// TIA Portal V18 export
TYPE "UDT_HCsDI"
// stored: IsFailsafeCompliant false
   STRUCT
      xHCPump1Ready : Array[1..2] of Bool;
      xHCPump1Ind : Array[1..2] of Bool;
      xHCPump1Alarm : Array[1..2] of Bool;
      xHCPump2Ready : Array[1..2] of Bool;
      xHCPump2Ind : Array[1..2] of Bool;
      xHCPump2Alarm : Array[1..2] of Bool;
      xHCDoublePumpInAuto : Array[1..2] of Bool;
   END_STRUCT;
   // xHCPump1Ready[1..2] := true;
   // xHCPump2Ready[1..2] := true;
END_TYPE
